PROGRAM PLC_Task_01
VAR
END_VAR

PRG_SL3L0_SCATTER();

END_PROGRAM

(* stored: Version 1.1.0.1, ProductVersion 3.1.4022.18
   POU PLC_Task_01: Id {03b7c84f-3d60-4e89-8483-adffb0dbdaa0}, SpecialFunc None *)
